PROGRAM MAIN
VAR
	FB_Test1		: FB_HeatingLoop;
	
	rPID_Core		: REAL;
	rPID_SUrface	: REAL;
	abIN_HE_Fault	: ARRAY [1..12] OF BOOL;
	
	iT_Core			: INT;
	iT_Surface		: INT;
	rmA				: REAL;
	bCore_Fault		: BOOL;
	bSurface_Fault	: BOOL;
	abOUT_HE_Fault	: ARRAY [1..12] OF BOOL;
END_VAR

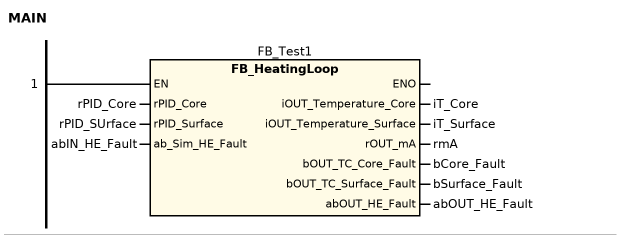
// NETWORK 1
FB_Test1(
    rPID_Core := rPID_Core,
    rPID_Surface := rPID_SUrface,
    ab_Sim_HE_Fault := abIN_HE_Fault,
    iOUT_Temperature_Core => iT_Core,
    iOUT_Temperature_Surface => iT_Surface,
    rOUT_mA => rmA,
    bOUT_TC_Core_Fault => bCore_Fault,
    bOUT_TC_Surface_Fault => bSurface_Fault,
    abOUT_HE_Fault => abOUT_HE_Fault); // FB_HeatingLoop

END_PROGRAM

(* stored: Version 1.1.0.1, ProductVersion 3.1.4024.12
   POU MAIN: Id {92689b9e-ea59-4841-8104-05164f048759}, SpecialFunc None *)
